// TwinCAT 3 PLC project PickAndPlacePlc
// ProgramVersion: 3.1.4024.0
// libraries:
//   Tc2_Standard, * (Beckhoff Automation GmbH)
//   Tc2_System, * (Beckhoff Automation GmbH)
//   Tc2_TcpIp, * (Beckhoff Automation GmbH)
//   Tc3_Module, * (Beckhoff Automation GmbH)
// project tree:
//   DUTs/PickAndPlaceUnit/ eSensorType.TcDUT (not stored), eSmPickAndPlace.TcDUT (not stored)
//   DUTs/TcpExchange/ eTcpStateMachine.TcDUT
//   / PlcTask.TcTTO, TcpExchange.TcTTO
//   POUs/Pick%27n%27Place Sequence/Objects/ FB_Gripper.TcPOU (not stored), FB_LinearMotor.TcPOU (not stored), FB_Motor.TcPOU (not stored), FB_Sensor.TcPOU (not stored)
//   POUs/Pick%27n%27Place Sequence/ PickAndPlaceUnit.TcPOU (not stored)
//   POUs/Pick%27n%27Place Sequence/Simulation/ FB_SensorsSimulation.TcPOU (not stored)
//   POUs/TcpExchange/Objects/ FB_TCPCameraServer.TcPOU
//   POUs/TcpExchange/ TcpCameraExchange.TcPOU
// real-time tasks:
//   TASK PlcTask: cycle T#10ms, priority 20, ADS port 350
//   TASK TcpExchange: cycle T#1ms, priority 1, ADS port 351

CONFIGURATION PickAndPlacePlc
    RESOURCE PLC ON TwinCAT3
        TASK PlcTask(INTERVAL := T#10ms, PRIORITY := 20);
        TASK TcpExchange(INTERVAL := T#1ms, PRIORITY := 1);
        PROGRAM PickAndPlaceUnit WITH PlcTask : PickAndPlaceUnit;
        PROGRAM TcpCameraExchange WITH TcpExchange : TcpCameraExchange;
    END_RESOURCE
END_CONFIGURATION

// ---- DUTs/TcpExchange/eTcpStateMachine.TcDUT
{attribute 'qualified_only'}
{attribute 'strict'}
TYPE eTcpStateMachine :
(
	INIT := 0,
	OPEN_SOCKET_LISTENER,
	ACCEPT_CLIENT_CONNECTION,
	RECEIVE_DATA,
	SEND_DATA,
	ERROR_HANDLING
	
	
);
END_TYPE

// ---- POUs/TcpExchange/TcpCameraExchange.TcPOU
PROGRAM TcpCameraExchange
VAR
	bInit: BOOL := TRUE;
	
	fbSocketCloseAll: FB_SocketCloseAll;                                // FB to close all sockets after login PLC with  download
	bSocketCloseError: BOOL;											
	nSocketCloseError: UDINT;
	
	fbTcpCameraServer: FB_TCPCameraServer;								// TCP server for camera data exchange

	bSignOfLife: BOOL;													// Send data status bit which changes every 500 ms
	fbSignOfLifeTmr: TON;												// Timer to change send data status bit

	udiValueToSend: UDINT;                                              // Value for camera
	udiSendData: UDINT;													// Data for camera to send with sign of life bit
	udiReceivedData: UDINT;												// Data from camera
	

	
	bStartServerCommunication: BOOL;									//
	bServerConnected: BOOL;
	bServerBusy: BOOL;
	bServerError: BOOL;
	nServerErrorID: UDINT;
END_VAR

VAR CONSTANT
	TCP_SIGN_OF_LIFE_PERIOD: TIME := T#500MS;
	TCP_POOL_TIME: TIME := T#100MS;
	TCP_SERVER_IP: T_IPv4Addr := '127.0.0.1';
	TCP_PORT_NUMBER: UDINT := 2010;
END_VAR


IF bInit THEN 	  												         // Close all sockets after login PLC with  download
	fbSocketCloseAll(
		sSrvNetId:= '', 
		bExecute:= TRUE, 
		tTimeout:= T#3S, 
		bBusy=> , 
		bError=> bSocketCloseError, 
		nErrId=> nSocketCloseError);
	IF NOT (fbSocketCloseAll.bBusy OR fbSocketCloseAll.bError) THEN
		bInit := FALSE;
		fbSocketCloseAll(bExecute:= FALSE);
	END_IF
ELSE		
	udiSendData := SHL(udiValueToSend,1);                               // Set value to send
	
	{region 'Adding sign of life bit to the data'}						// Add sign of life bit
	fbSignOfLifeTmr(IN:= NOT fbSignOfLifeTmr.Q, 
					PT:= TCP_SIGN_OF_LIFE_PERIOD, 
					Q=> , 
					ET=> );
	IF fbSignOfLifeTmr.Q THEN
		bSignOfLife := NOT bSignOfLife;		
	END_IF;	
	udiSendData.0 := bSignOfLife;	 
	{endregion}
	
	{region 'TCP server fb call'}										//
	fbTcpCameraServer(
		sLocalHost:= TCP_SERVER_IP, 									// Server IP Adress
		nLocalPort:= TCP_PORT_NUMBER, 									// Server port
		tPoolTime:= TCP_POOL_TIME,
		bStartCommunication:= bStartServerCommunication, 				// Allow Client-connection or close connection
		udiSendData:= udiSendData,
		bConnected => bServerConnected,									// Client connection is valid
		udiReceivedData => udiReceivedData,
		bBusy=> bServerBusy, 
		bError=> bServerError, 
		nErrorID=> nServerErrorID);
END_IF

END_PROGRAM

// ---- POUs/TcpExchange/Objects/FB_TCPCameraServer.TcPOU
FUNCTION_BLOCK FB_TCPCameraServer
VAR_INPUT
	sLocalHost: T_IPv4Addr;											// Server IP address
	nLocalPort: UDINT;												// Server port number
	tPoolTime: TIME;												// Pool time for data exchange
	bStartCommunication : BOOL;										// Start the exchange process
	udiSendData: UDINT;												// Data to send to client
END_VAR
VAR_OUTPUT
	bConnected: BOOL;												// Client connection is accepted
	udiReceivedData: UDINT;											// Data received from client
	bBusy: BOOL;													
	bError: BOOL;
	nErrorID: UDINT;
END_VAR
VAR
	iState: eTcpStateMachine;
	hListener: T_HSOCKET;                                           // Handler from socket listener
	hSocket: T_HSOCKET;												// Handler from remote client accept
	
	fbSocketListen: FB_SocketListen;								// Open socket listener
	fbSocketAccept: FB_SocketAccept;								// Accept remote client connection
	fbSocketSend: FB_SocketSend;									// Send data to socket
	fbSocketReceive: FB_SocketReceive;								// Receive data to socket
	fbSocketClose: FB_SocketClose;									// Close socket
	
	bSendTrigger: BOOL;												// Cyclical trigger to send data to client
	fbPoolTmr: TON;													// Timer to produce send command
	
END_VAR

CASE iState OF

	eTcpStateMachine.INIT: 											// SM: Init State, reinitialize FBs
	
		IF bStartCommunication = TRUE THEN							// If communication was started
			fbSocketListen(bExecute := FALSE);						// Reinitialize	socket listener FB
			fbSocketAccept(bExecute := FALSE);						// Reinitialize	remote client connection acceptance FB
			fbSocketClose(bExecute:= FALSE);						// Reinitialize	socket close FB
			bBusy := TRUE;				
			iState := eTcpStateMachine.OPEN_SOCKET_LISTENER;		// Activate OPEN_SOCKET_LISTENER
		ELSE
			bBusy := FALSE;
		END_IF
	
		
	eTcpStateMachine.OPEN_SOCKET_LISTENER:							// SM: Open socket listener
	
		fbSocketListen(sSrvNetId:= '', 								// NetID for local server
					   sLocalHost:= sLocalHost, 					// Local IP address
					   nLocalPort:= nLocalPort, 					// Local Port number
					   bExecute:= TRUE, 
					   tTimeout:= T#4S, 
					   bBusy=> , 
					   bError=> bError, 
					   nErrId=> nErrorID,
					   hListener=> hListener);						// Handle to send and receive data from socket
		
		IF hListener.handle <> 0 THEN								// If socket was opened succsessfully
			iState :=eTcpStateMachine.ACCEPT_CLIENT_CONNECTION;		// Activate ACCEPT_CLIENT_CONNECTION step
		ELSIF bError THEN
			iState := eTcpStateMachine.ERROR_HANDLING;				// Activate ERROR_HANDLING
		END_IF
	
		
	eTcpStateMachine.ACCEPT_CLIENT_CONNECTION: 						// Accept remote client connection
	
		fbSocketAccept(sSrvNetId:= '', 		
					   hListener:= hListener, 				    	// Handle from socket listener
					   bExecute:= TRUE, 
					   tTimeout:= T#4S, 
					   bAccepted=> , 
					   bBusy=> , 
					   bError=> bError, 
				       nErrId=> nErrorID,
					   hSocket=> hSocket);							// Connection handle
		
		IF NOT fbSocketAccept.bBusy THEN
			fbSocketAccept(bExecute:= FALSE);
		END_IF

		IF hSocket.handle <> 0 THEN									// Client connection was accepted
			iState := eTcpStateMachine.SEND_DATA;					// Activate SEND_DATA
			bConnected := TRUE;										// Change "Connected" status
		ELSIF bError THEN									
			iState := eTcpStateMachine.ERROR_HANDLING; 				// Activate ERROR_HANDLING
		END_IF


	eTcpStateMachine.SEND_DATA: 									// SM: Send Data
	
		fbPoolTmr(IN:= NOT fbPoolTmr.Q, 							// Pool tmr to send data
				  PT:= tPoolTime, 
				  Q=> , 
				  ET=> );	
				  
		fbSocketSend(sSrvNetId:= '', 								// Send data to client with pool period
					 hSocket:= hSocket, 							// Handle from socket accept
					 cbLen:= SIZEOF(udiSendData), 
					 pSrc:= ADR(udiSendData),
					 bExecute:= fbPoolTmr.Q, 
					 tTimeout:= T#3S, 
					 bBusy=> , 
					 bError=> bError, 
					 nErrId=> nErrorID);		
	
		IF NOT fbSocketSend.bBusy THEN						   		// Switch back to receiving state after sending
			iState := eTcpStateMachine.RECEIVE_DATA;		   		// Close connection in case of error 
		END_IF
		IF fbSocketSend.bError OR(NOT bStartCommunication) THEN  // Close connection when error is occuring or trigger is set
			iState := eTcpStateMachine.ERROR_HANDLING;				// Activate ERROR_HANDLING
		END_IF
		
	
		
	eTcpStateMachine.RECEIVE_DATA: 									// SM: Receive Data

		fbSocketReceive(sSrvNetId:= '', 							// Check cyclically for new data from client
						hSocket:= hSocket, 							// Handle from socket accept
						cbLen:= SIZEOF(udiReceivedData), 
						pDest:= ADR(udiReceivedData), 
						bExecute:= TRUE, 														
						tTimeout:= T#4S, 
						bBusy=> , 
						bError=> bError, 
						nErrId=> nErrorID,
						nRecBytes=> );
		
		IF NOT fbSocketReceive.bBusy THEN							// If the data was received successfully
			fbSocketReceive(bExecute := FALSE);						
			iState := eTcpStateMachine.SEND_DATA;					// Activate SEND_DATA
		END_IF
		IF fbSocketReceive.bError OR(NOT bStartCommunication) THEN  // Close connection when error is occuring or trigger is set
			iState := eTcpStateMachine.ERROR_HANDLING;				// Activate ERROR_HANDLING
		END_IF


	eTcpStateMachine.ERROR_HANDLING:								// SM: Error Handling	

		fbSocketClose(sSrvNetId:= '', 								// Close socket listener
					  hSocket:= hListener, 
					  bExecute:= TRUE, 
					  tTimeout:= T#4S, 
					  bBusy=> , 
					  bError=> bError, 
					  nErrId=> nErrorID);		

		fbSocketClose(sSrvNetId:= '', 								// Close socket client connection
					  hSocket:= hSocket, 
					  bExecute:= TRUE, 
					  tTimeout:= T#4S, 
					  bBusy=> , 
					  bError=> bError, 
					  nErrId=> nErrorID);
					  
		IF NOT (fbSocketClose.bBusy) OR fbSocketClose.bError THEN   // If socket is closed
			hSocket.handle := 0;	
			iState := eTcpStateMachine.INIT;						// Activate INIT
			bConnected := FALSE;
		END_IF
	
END_CASE

END_FUNCTION_BLOCK
